Fanuc KAREL source: f_attr_t.kl

PROGRAM F_ATTR_T
%ALPHABETIZE
%CMOSVARS
%COMMENT = 'test attr'
%CRTDEVICE
%DEFGROUP = 1
%DELAY = 10
%ENVIRONMENT TPE
%NOABORT = ERROR + COMMAND
%NOBUSYLAMP
%NOLOCKGROUP
%NOPAUSE = ERROR + COMMAND + TPENABLE
%NOPAUSESHFT
%PRIORITY = 60
%STACKSIZE = 600
%TIMESLICE = 32
%TPMOTION
%SYSTEM
%INVISIBLE
VAR
  zz, aa : INTEGER
BEGIN
  zz = 1
END F_ATTR_T
